// TIA Portal V17 export
// export: Created 2022-03-12T16:05:28.7879569Z, ExportSetting WithDefaults, DisplayName Totally Integrated Automation Portal, DisplayVersion V17, DisplayName TIA Portal Openness, DisplayVersion V17, DisplayName TIA Portal Version Control Interface, DisplayVersion V17, DisplayName STEP 7 Professional, DisplayVersion V17, DisplayName STEP 7 Safety, DisplayVersion V17, DisplayName WinCC Advanced / Unified PC, DisplayVersion V17
DATA_BLOCK "InstEM01_00_Main"   // DB31660
TITLE = InstEM01_00_Main
AUTHOR : tech.team.motioncontrol@siemens.com
FAMILY : CPG
VERSION : 1.0
// Support: tech.team.motioncontrol@siemens.com
// Fax: +49 (0) 9131/98-1297
// stored: AutoNumber true, DBAccessibleFromOPCUA true, DBAccessibleFromWebserver true, InstanceOfName EM01_00_Main, InstanceOfType FB
"EM01_00_Main"
   // VAR
   //    instEventControl { ExternalAccessible := 'False'; ExternalVisible := 'False'; ExternalWritable := 'False'; S7_SetPoint := 'True'} : "EM01_01_EventControl";
   //    instPackML_ModuleSum { ExternalAccessible := 'False'; ExternalVisible := 'False'; ExternalWritable := 'False'; S7_SetPoint := 'True'} : "EM01_02_PackML_ModuleSum";
   //    instCM01 { ExternalAccessible := 'False'; ExternalVisible := 'False'; ExternalWritable := 'False'; S7_SetPoint := 'True'} : "EM01_CM01_Conveyor";
   //    instCM02 { ExternalAccessible := 'False'; ExternalVisible := 'False'; ExternalWritable := 'False'; S7_SetPoint := 'True'} : "EM01_CM02_Palletizer";
   // END_VAR
BEGIN
END_DATA_BLOCK
